(* PLC project Unnamed, Unknown Unnamed 1 *)
(* stored: creationDateTime 2024-11-27T13:15:33, modificationDateTime 2024-12-24T00:01:56 *)

PROGRAM program0
  VAR
    S1 : BOOL;  (* Push Button S1 *)
    x : BOOL;
    Reset : BOOL;  (* Reset *)
    Actual_Input_Signal : BOOL;  (* Used because S1 is non-latching *)
    Cylinder_2 : BOOL;  (* If True,cylinder is forward *)
    B7 : BOOL;  (* Signals the presence of part *)
    Cylinder_1 : BOOL;  (* If True,cylinder is forward *)
    B2 : BOOL;  (* Cylinder-1 is forward *)
    y : BOOL;  (* If True,cylinder 1 retracts. *)
    B3 : BOOL;  (* Cylinder-2 is retracted *)
    B4 : BOOL;  (* Cylinder-2 is forward *)
    B5 : BOOL;  (* Cylinder-3 is retracted *)
    B6 : BOOL;  (* Cylinder-3 is forward *)
    Cylinder_3 : BOOL;  (* If True,cylinder is forward *)
    CTU0 : CTU;
    CTU1 : CTU;
    TOF0 : TOF;
    CTU2 : CTU;
    TON1 : TON;
    TON0 : TON;
  END_VAR
  VAR  (* added by the conversion: wires and edge detectors of the diagram *)
    _XOR60_OUT : BOOL;
    R_TRIG1 : R_TRIG;
    R_TRIG2 : R_TRIG;
    _AND40_OUT : BOOL;
    R_TRIG3 : R_TRIG;
  END_VAR

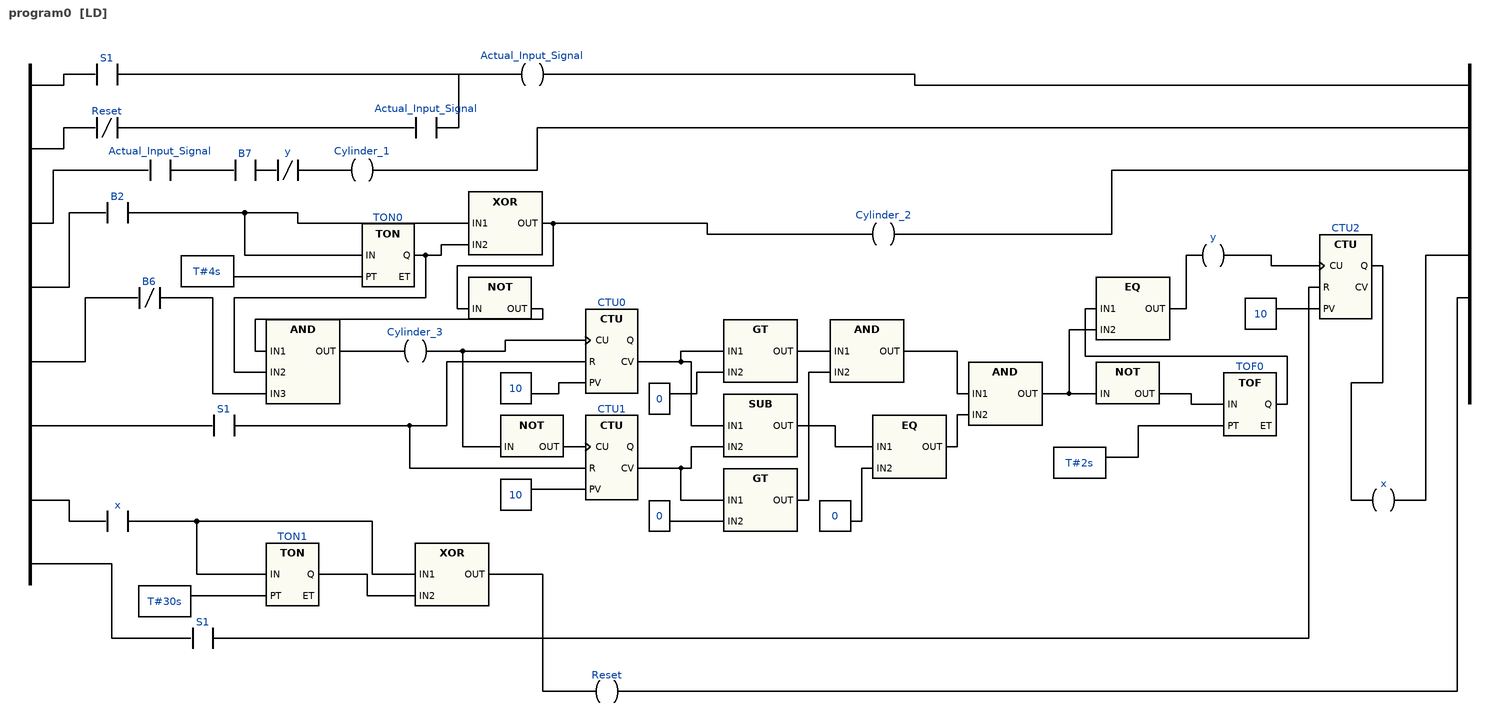
(* LD diagram, written out as Structured Text *)
Cylinder_1 := Actual_Input_Signal AND B7 AND NOT y;
Actual_Input_Signal := S1 OR NOT Reset AND Actual_Input_Signal;
TON0(IN := B2, PT := T#4s);
_XOR60_OUT := B2 XOR TON0.Q;
R_TRIG1(CLK := NOT _XOR60_OUT AND TON0.Q AND NOT B6);
CTU0(CU := R_TRIG1.Q, R := S1, PV := 10);
R_TRIG2(CLK := NOT (NOT _XOR60_OUT AND TON0.Q AND NOT B6));
CTU1(CU := R_TRIG2.Q, R := S1, PV := 10);
_AND40_OUT := CTU0.CV > 0 AND CTU1.CV > 0 AND CTU0.CV - CTU1.CV = 0;
TOF0(IN := NOT _AND40_OUT, PT := T#2s);
y := TOF0.Q = _AND40_OUT;
R_TRIG3(CLK := TOF0.Q = _AND40_OUT);
CTU2(CU := R_TRIG3.Q, R := S1, PV := 10);
x := CTU2.Q;
TON1(IN := x, PT := T#30s);
Reset := x XOR TON1.Q;
Cylinder_2 := _XOR60_OUT;
Cylinder_3 := NOT _XOR60_OUT AND TON0.Q AND NOT B6;
END_PROGRAM

CONFIGURATION Config0
  RESOURCE Res0 ON PLC
    TASK task0(INTERVAL := T#20ms, PRIORITY := 0);
    PROGRAM instance0 WITH task0 : program0;
  END_RESOURCE
END_CONFIGURATION
